FUNCTION_BLOCK IN_OUT_DIS_PRESS_BUTTON (* Button with boolean input display from controller and events on each press / release *)
  (* Standard: 61499-2 *)
  (* Version 1.0, 2006-01-05, Anirudha, UoA, Corrected output event *)
  (* Version 0.2, 2005-12-04, Anirudha, UoA, Added colors *)
  (* Compiler header: package fb.rt.vhmi; *)
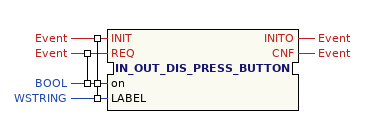
  EVENT_INPUT
    INIT WITH on, LABEL; (* Initialization Request *)
    REQ WITH on; (* Normal Execution Request *)
  END_EVENT
  EVENT_OUTPUT
    INITO; (* Initialization Confirm *)
    CNF; (* Execution Confirmation *)
  END_EVENT
  VAR_INPUT
    on : BOOL;
    LABEL : WSTRING;
  END_VAR
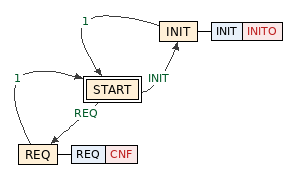
  EC_STATES
    START; (* Initial State *)
    INIT : INIT -> INITO; (* Initialization *)
    REQ : REQ -> CNF; (* Normal execution *)
  END_STATES
  EC_TRANSITIONS
    START TO INIT := INIT;
    INIT TO START := 1;
    START TO REQ := REQ;
    REQ TO START := 1;
  END_TRANSITIONS
  ALGORITHM INIT IN ST: (* Initialization algorithm *)

  END_ALGORITHM
  ALGORITHM REQ IN ST: (* Normally executed algorithm *)

  END_ALGORITHM
END_FUNCTION_BLOCK
